INTERFACE I_InterfaceDatatypeAddedEvent EXTENDS I_Event

PROPERTY PUBLIC Target : I_InterfaceDatatype
GET
END_GET
END_PROPERTY

END_INTERFACE

(* stored: Version 1.1.0.1, ProductVersion 3.1.4024.12
   Itf I_InterfaceDatatypeAddedEvent: Id {bc6eada9-8af1-4b92-8dab-a08824ed4677}
   Property Target: Id {1124cc2b-e868-44f1-a6d2-ee20f20db975}
   Get Get: Id {64690bd8-c0b8-46f3-9c8e-054e9a672b70} *)
